(* Schneider Machine Expert - Basic project Comparação de valores IO analógicas, file version 3.0.0.0 *)
(* ProjectInformations: Name=Novo projeto *)

HARDWARE
  Cpu 0: TM221CE40R
  EthernetConfiguration: NetworkName=M221, IpAllocationMode=FixedAddress, IpAddress=0.0.0.0, SubnetMask=0.0.0.0
  SerialLineConfiguration: Baud=Baud19200, Parity=ParityEven, DataBits=DataBits8, StopBits=StopBits1, PhysicalMedium=PhysicalMediumRs485, TransmissionMode=TransmissionModeModbusRtu, SlaveId=1, Addressing=SlaveAddressing
  MastTask: UsePeriodScanMode=false, PeriodScan=100
  FastTask: Period=255
  CpuBehavior: StartingMode=StartAsPreviousState, AutoSaveRamOnEeprom=true, WatchdogPeriod=250

SYMBOLS  (address, symbol, comment, settings)
  %IW0.0      [Type=Type_0_10V, Scope=Scope_Normal, Minimum=0, Maximum=1000]

POU Novo POU
  (* SectionNumber=1 *)

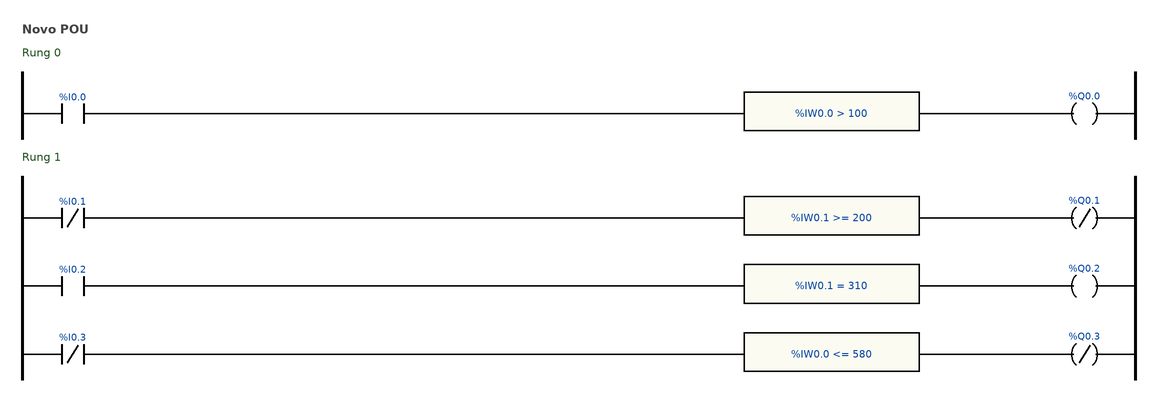

// Rung 0
  LD %I0.0
  AND [ %IW0.0 > 100 ]
  ST %Q0.0
  // as ST:
  //   %Q0.0 := %I0.0 AND %IW0.0 > 100;

// Rung 1
  (* no IL stored for this rung *)
